TYPE ST_AnalogInputDiag :
STRUCT
	Underrange			: BIT;
	Overrange			: BIT;
	Error				: BIT;
END_STRUCT 
END_TYPE

(* stored: Version 1.1.0.1, ProductVersion 3.1.4026.18
   DUT ST_AnalogInputDiag: Id {763bb98d-e860-4492-a00f-edeacf183cb7} *)
